// TIA Portal V17 export
// export: Created 2025-04-25T10:07:02.8968061Z, ExportSetting WithDefaults, DisplayName Totally Integrated Automation Portal, DisplayVersion V17 Update 8, DisplayName TIA Portal Openness, DisplayVersion V17 Update 8, DisplayName TIA Portal Version Control Interface, DisplayVersion V17, DisplayName SINAMICS Startdrive Advanced, DisplayVersion V17 SP2, DisplayName SINAMICS Startdrive G110M, G120, G120C, G120D, G120P, G115D, DisplayVersion V17 SP2, DisplayName SINAMICS Startdrive G130, G150, S120, S150, SINAMICS MV, S210, DisplayVersion V17 SP2, DisplayName STEP 7 Professional, DisplayVersion V17 Update 8, DisplayName SINUMERIK ONE STEP 7 Toolbox, DisplayVersion V17 Update 12, DisplayName SINUMERIK 840D sl STEP 7 Toolbox, DisplayVersion V17 Update 12, DisplayName STEP 7 Safety, DisplayVersion V17 Update 6, DisplayName WinCC Advanced / Unified PC, DisplayVersion V17 Update 8
FUNCTION "FC7342_MACHINE_TO_POWDER_PLC_INTERLOCK" : Void   // FC7342, LAD
{ S7_Optimized_Access := 'TRUE' }
VERSION : 0.1
// stored: AutoNumber false, IsIECCheckEnabled false, SetENOAutomatically false, UDAEnableTagReadback false
   VAR_TEMP
      RET_VAL_1 : Int;
   END_VAR
BEGIN

REGION Network 1: LIFE BIT
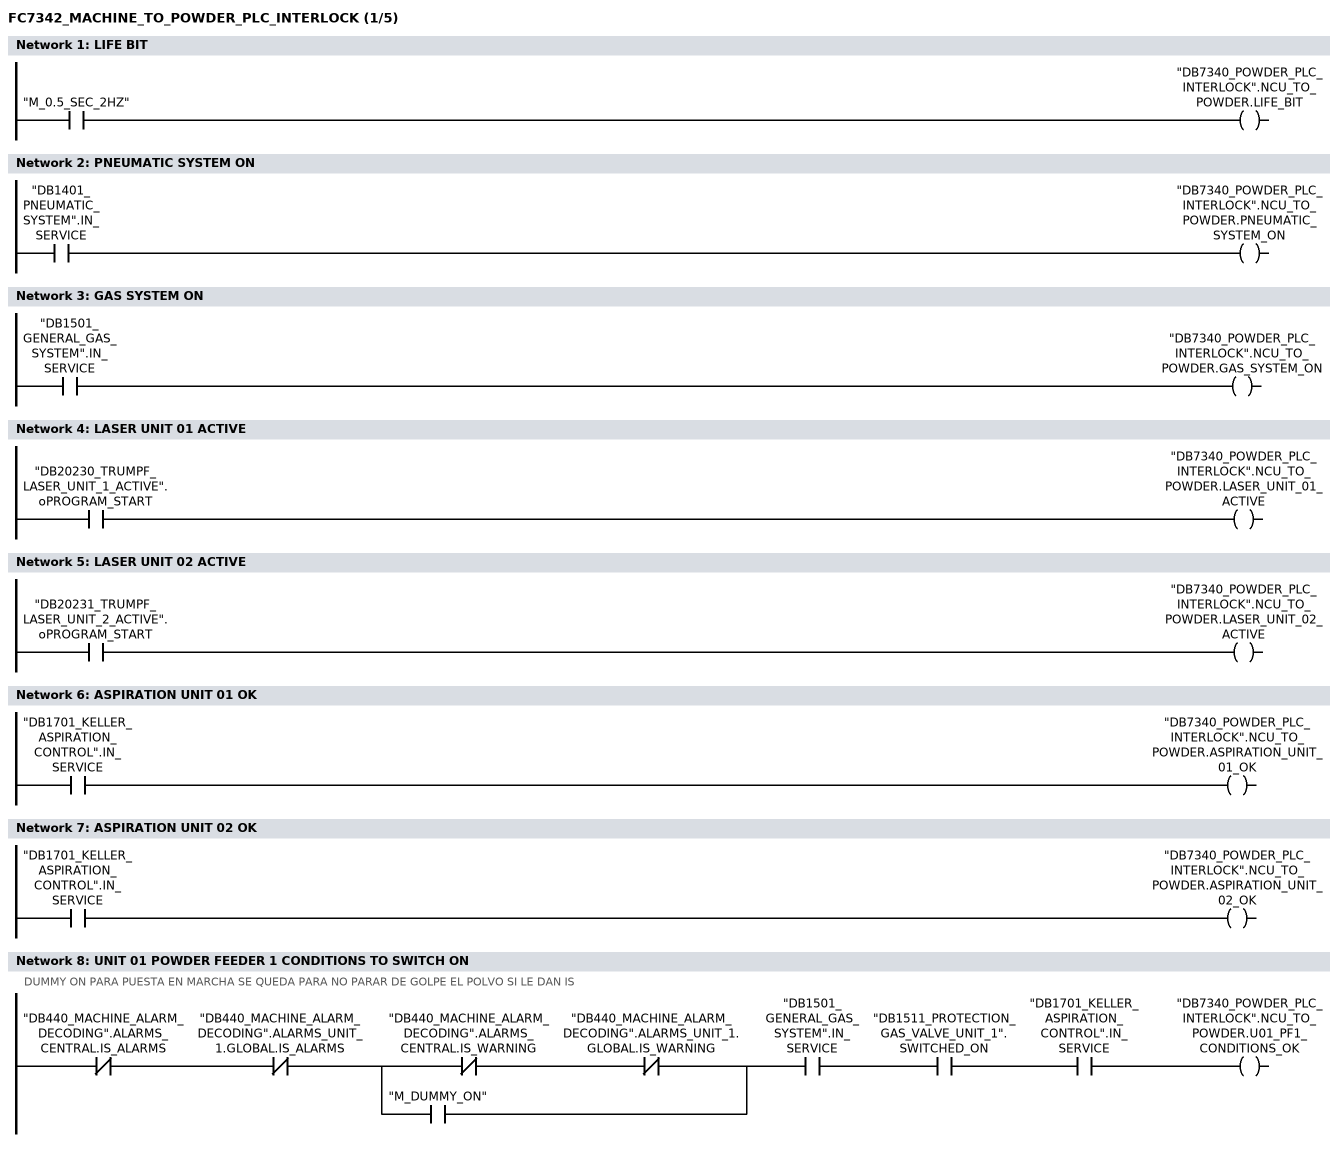
   RUNG wire#powerrail
      Contact( "M_0.5_SEC_2HZ" )
      Coil( "DB7340_POWDER_PLC_INTERLOCK".NCU_TO_POWDER.LIFE_BIT )
   END_RUNG
   // the same network as SCL:
   "DB7340_POWDER_PLC_INTERLOCK".NCU_TO_POWDER.LIFE_BIT := "M_0.5_SEC_2HZ";
END_REGION

REGION Network 2: PNEUMATIC SYSTEM ON
   RUNG wire#powerrail
      Contact( "DB1401_PNEUMATIC_SYSTEM".IN_SERVICE )
      Coil( "DB7340_POWDER_PLC_INTERLOCK".NCU_TO_POWDER.PNEUMATIC_SYSTEM_ON )
   END_RUNG
   // the same network as SCL:
   "DB7340_POWDER_PLC_INTERLOCK".NCU_TO_POWDER.PNEUMATIC_SYSTEM_ON := "DB1401_PNEUMATIC_SYSTEM".IN_SERVICE;
END_REGION

REGION Network 3: GAS SYSTEM ON
   RUNG wire#powerrail
      Contact( "DB1501_GENERAL_GAS_SYSTEM".IN_SERVICE )
      Coil( "DB7340_POWDER_PLC_INTERLOCK".NCU_TO_POWDER.GAS_SYSTEM_ON )
   END_RUNG
   // the same network as SCL:
   "DB7340_POWDER_PLC_INTERLOCK".NCU_TO_POWDER.GAS_SYSTEM_ON := "DB1501_GENERAL_GAS_SYSTEM".IN_SERVICE;
END_REGION

REGION Network 4: LASER UNIT 01 ACTIVE
   RUNG wire#powerrail
      Contact( "DB20230_TRUMPF_LASER_UNIT_1_ACTIVE".oPROGRAM_START )
      Coil( "DB7340_POWDER_PLC_INTERLOCK".NCU_TO_POWDER.LASER_UNIT_01_ACTIVE )
   END_RUNG
   // the same network as SCL:
   "DB7340_POWDER_PLC_INTERLOCK".NCU_TO_POWDER.LASER_UNIT_01_ACTIVE := "DB20230_TRUMPF_LASER_UNIT_1_ACTIVE".oPROGRAM_START;
END_REGION

REGION Network 5: LASER UNIT 02 ACTIVE
   RUNG wire#powerrail
      Contact( "DB20231_TRUMPF_LASER_UNIT_2_ACTIVE".oPROGRAM_START )
      Coil( "DB7340_POWDER_PLC_INTERLOCK".NCU_TO_POWDER.LASER_UNIT_02_ACTIVE )
   END_RUNG
   // the same network as SCL:
   "DB7340_POWDER_PLC_INTERLOCK".NCU_TO_POWDER.LASER_UNIT_02_ACTIVE := "DB20231_TRUMPF_LASER_UNIT_2_ACTIVE".oPROGRAM_START;
END_REGION

REGION Network 6: ASPIRATION UNIT 01 OK
   RUNG wire#powerrail
      Contact( "DB1701_KELLER_ASPIRATION_CONTROL".IN_SERVICE )
      Coil( "DB7340_POWDER_PLC_INTERLOCK".NCU_TO_POWDER.ASPIRATION_UNIT_01_OK )
   END_RUNG
   // the same network as SCL:
   "DB7340_POWDER_PLC_INTERLOCK".NCU_TO_POWDER.ASPIRATION_UNIT_01_OK := "DB1701_KELLER_ASPIRATION_CONTROL".IN_SERVICE;
END_REGION

REGION Network 7: ASPIRATION UNIT 02 OK
   RUNG wire#powerrail
      Contact( "DB1701_KELLER_ASPIRATION_CONTROL".IN_SERVICE )
      Coil( "DB7340_POWDER_PLC_INTERLOCK".NCU_TO_POWDER.ASPIRATION_UNIT_02_OK )
   END_RUNG
   // the same network as SCL:
   "DB7340_POWDER_PLC_INTERLOCK".NCU_TO_POWDER.ASPIRATION_UNIT_02_OK := "DB1701_KELLER_ASPIRATION_CONTROL".IN_SERVICE;
END_REGION

REGION Network 8: UNIT 01 POWDER FEEDER 1 CONDITIONS TO SWITCH ON
   // DUMMY ON PARA PUESTA EN MARCHA SE QUEDA PARA NO PARAR DE GOLPE EL POLVO SI LE DAN IS
   RUNG wire#powerrail
      I_Contact( "DB440_MACHINE_ALARM_DECODING".ALARMS_CENTRAL.IS_ALARMS )
      I_Contact( "DB440_MACHINE_ALARM_DECODING".ALARMS_UNIT_1.GLOBAL.IS_ALARMS )
      wire#w1
      I_Contact( "DB440_MACHINE_ALARM_DECODING".ALARMS_CENTRAL.IS_WARNING )
      I_Contact( "DB440_MACHINE_ALARM_DECODING".ALARMS_UNIT_1.GLOBAL.IS_WARNING )
      wire#w2
      Contact( "DB1501_GENERAL_GAS_SYSTEM".IN_SERVICE )
      Contact( "DB1511_PROTECTION_GAS_VALVE_UNIT_1".SWITCHED_ON )
      Contact( "DB1701_KELLER_ASPIRATION_CONTROL".IN_SERVICE )
      Coil( "DB7340_POWDER_PLC_INTERLOCK".NCU_TO_POWDER.U01_PF1_CONDITIONS_OK )
   END_RUNG
   RUNG wire#w1
      Contact( "M_DUMMY_ON" )
   END_RUNG wire#w2
   // the same network as SCL:
   "DB7340_POWDER_PLC_INTERLOCK".NCU_TO_POWDER.U01_PF1_CONDITIONS_OK := NOT "DB440_MACHINE_ALARM_DECODING".ALARMS_CENTRAL.IS_ALARMS AND NOT "DB440_MACHINE_ALARM_DECODING".ALARMS_UNIT_1.GLOBAL.IS_ALARMS AND ((NOT "DB440_MACHINE_ALARM_DECODING".ALARMS_CENTRAL.IS_WARNING AND NOT "DB440_MACHINE_ALARM_DECODING".ALARMS_UNIT_1.GLOBAL.IS_WARNING) OR "M_DUMMY_ON") AND "DB1501_GENERAL_GAS_SYSTEM".IN_SERVICE AND "DB1511_PROTECTION_GAS_VALVE_UNIT_1".SWITCHED_ON AND "DB1701_KELLER_ASPIRATION_CONTROL".IN_SERVICE;
END_REGION

REGION Network 9: UNIT 02 POWDER FEEDER 1 CONDITIONS TO SWITCH ON
   // DUMMY ON PARA PUESTA EN MARCHA SE QUEDA PARA NO PARAR DE GOLPE EL POLVO SI LE DAN IS
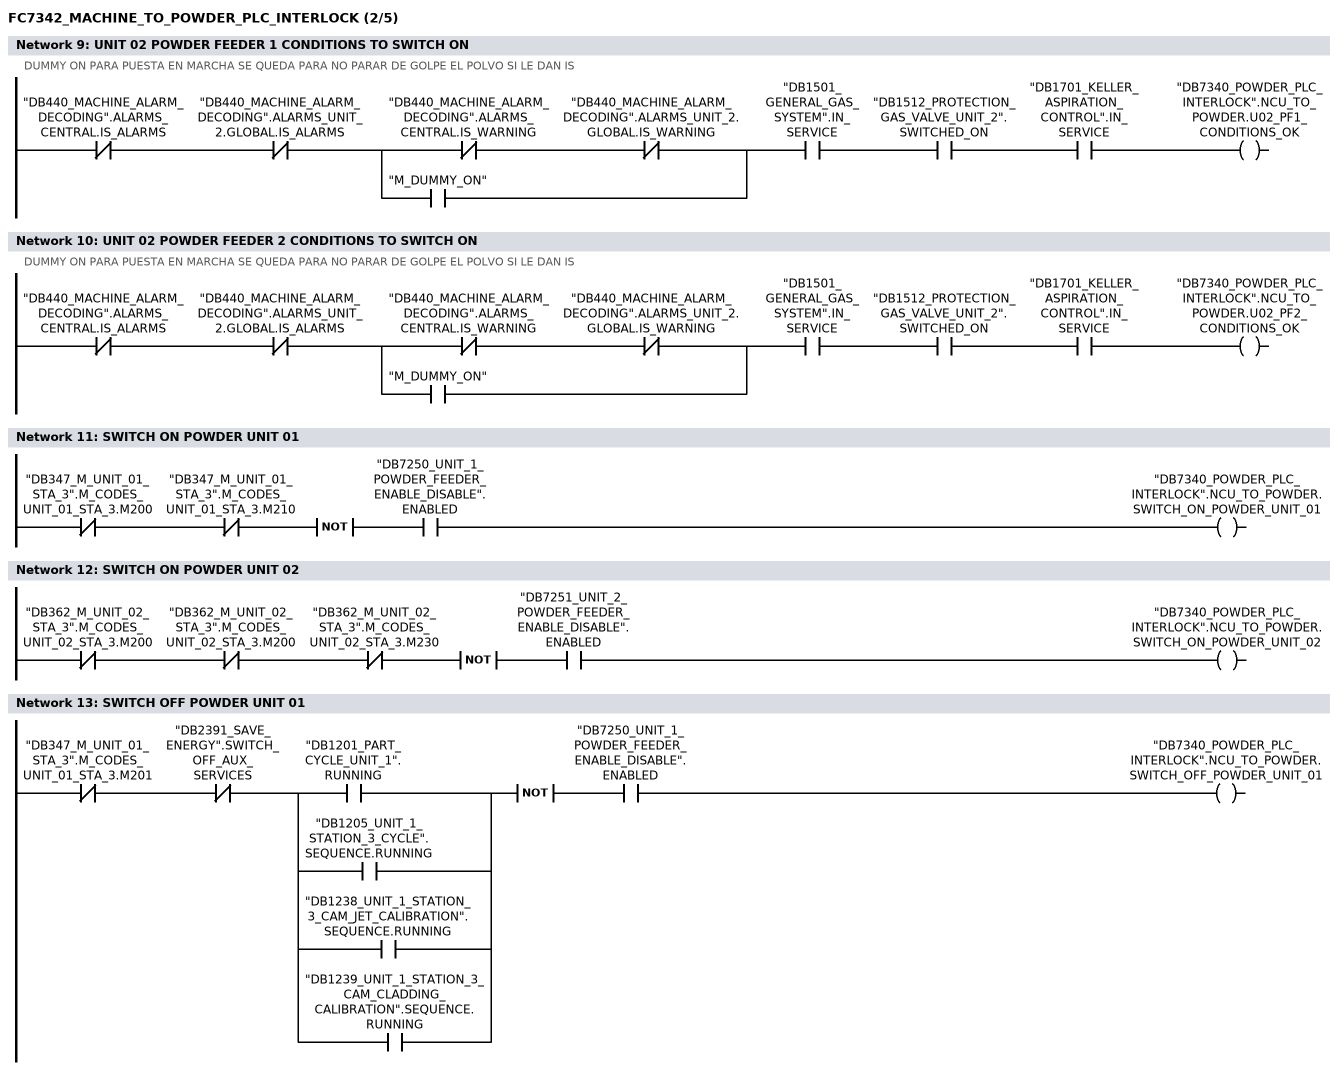
   RUNG wire#powerrail
      I_Contact( "DB440_MACHINE_ALARM_DECODING".ALARMS_CENTRAL.IS_ALARMS )
      I_Contact( "DB440_MACHINE_ALARM_DECODING".ALARMS_UNIT_2.GLOBAL.IS_ALARMS )
      wire#w1
      I_Contact( "DB440_MACHINE_ALARM_DECODING".ALARMS_CENTRAL.IS_WARNING )
      I_Contact( "DB440_MACHINE_ALARM_DECODING".ALARMS_UNIT_2.GLOBAL.IS_WARNING )
      wire#w2
      Contact( "DB1501_GENERAL_GAS_SYSTEM".IN_SERVICE )
      Contact( "DB1512_PROTECTION_GAS_VALVE_UNIT_2".SWITCHED_ON )
      Contact( "DB1701_KELLER_ASPIRATION_CONTROL".IN_SERVICE )
      Coil( "DB7340_POWDER_PLC_INTERLOCK".NCU_TO_POWDER.U02_PF1_CONDITIONS_OK )
   END_RUNG
   RUNG wire#w1
      Contact( "M_DUMMY_ON" )
   END_RUNG wire#w2
   // the same network as SCL:
   "DB7340_POWDER_PLC_INTERLOCK".NCU_TO_POWDER.U02_PF1_CONDITIONS_OK := NOT "DB440_MACHINE_ALARM_DECODING".ALARMS_CENTRAL.IS_ALARMS AND NOT "DB440_MACHINE_ALARM_DECODING".ALARMS_UNIT_2.GLOBAL.IS_ALARMS AND ((NOT "DB440_MACHINE_ALARM_DECODING".ALARMS_CENTRAL.IS_WARNING AND NOT "DB440_MACHINE_ALARM_DECODING".ALARMS_UNIT_2.GLOBAL.IS_WARNING) OR "M_DUMMY_ON") AND "DB1501_GENERAL_GAS_SYSTEM".IN_SERVICE AND "DB1512_PROTECTION_GAS_VALVE_UNIT_2".SWITCHED_ON AND "DB1701_KELLER_ASPIRATION_CONTROL".IN_SERVICE;
END_REGION

REGION Network 10: UNIT 02 POWDER FEEDER 2 CONDITIONS TO SWITCH ON
   // DUMMY ON PARA PUESTA EN MARCHA SE QUEDA PARA NO PARAR DE GOLPE EL POLVO SI LE DAN IS
   RUNG wire#powerrail
      I_Contact( "DB440_MACHINE_ALARM_DECODING".ALARMS_CENTRAL.IS_ALARMS )
      I_Contact( "DB440_MACHINE_ALARM_DECODING".ALARMS_UNIT_2.GLOBAL.IS_ALARMS )
      wire#w1
      I_Contact( "DB440_MACHINE_ALARM_DECODING".ALARMS_CENTRAL.IS_WARNING )
      I_Contact( "DB440_MACHINE_ALARM_DECODING".ALARMS_UNIT_2.GLOBAL.IS_WARNING )
      wire#w2
      Contact( "DB1501_GENERAL_GAS_SYSTEM".IN_SERVICE )
      Contact( "DB1512_PROTECTION_GAS_VALVE_UNIT_2".SWITCHED_ON )
      Contact( "DB1701_KELLER_ASPIRATION_CONTROL".IN_SERVICE )
      Coil( "DB7340_POWDER_PLC_INTERLOCK".NCU_TO_POWDER.U02_PF2_CONDITIONS_OK )
   END_RUNG
   RUNG wire#w1
      Contact( "M_DUMMY_ON" )
   END_RUNG wire#w2
   // the same network as SCL:
   "DB7340_POWDER_PLC_INTERLOCK".NCU_TO_POWDER.U02_PF2_CONDITIONS_OK := NOT "DB440_MACHINE_ALARM_DECODING".ALARMS_CENTRAL.IS_ALARMS AND NOT "DB440_MACHINE_ALARM_DECODING".ALARMS_UNIT_2.GLOBAL.IS_ALARMS AND ((NOT "DB440_MACHINE_ALARM_DECODING".ALARMS_CENTRAL.IS_WARNING AND NOT "DB440_MACHINE_ALARM_DECODING".ALARMS_UNIT_2.GLOBAL.IS_WARNING) OR "M_DUMMY_ON") AND "DB1501_GENERAL_GAS_SYSTEM".IN_SERVICE AND "DB1512_PROTECTION_GAS_VALVE_UNIT_2".SWITCHED_ON AND "DB1701_KELLER_ASPIRATION_CONTROL".IN_SERVICE;
END_REGION

REGION Network 11: SWITCH ON POWDER UNIT 01
   RUNG wire#powerrail
      I_Contact( "DB347_M_UNIT_01_STA_3".M_CODES_UNIT_01_STA_3.M200 )
      I_Contact( "DB347_M_UNIT_01_STA_3".M_CODES_UNIT_01_STA_3.M210 )
      Not()
      Contact( "DB7250_UNIT_1_POWDER_FEEDER_ENABLE_DISABLE".ENABLED )
      Coil( "DB7340_POWDER_PLC_INTERLOCK".NCU_TO_POWDER.SWITCH_ON_POWDER_UNIT_01 )
   END_RUNG
   // the same network as SCL:
   "DB7340_POWDER_PLC_INTERLOCK".NCU_TO_POWDER.SWITCH_ON_POWDER_UNIT_01 := NOT (NOT "DB347_M_UNIT_01_STA_3".M_CODES_UNIT_01_STA_3.M200 AND NOT "DB347_M_UNIT_01_STA_3".M_CODES_UNIT_01_STA_3.M210) AND "DB7250_UNIT_1_POWDER_FEEDER_ENABLE_DISABLE".ENABLED;
END_REGION

REGION Network 12: SWITCH ON POWDER UNIT 02
   RUNG wire#powerrail
      I_Contact( "DB362_M_UNIT_02_STA_3".M_CODES_UNIT_02_STA_3.M200 )
      I_Contact( "DB362_M_UNIT_02_STA_3".M_CODES_UNIT_02_STA_3.M200 )
      I_Contact( "DB362_M_UNIT_02_STA_3".M_CODES_UNIT_02_STA_3.M230 )
      Not()
      Contact( "DB7251_UNIT_2_POWDER_FEEDER_ENABLE_DISABLE".ENABLED )
      Coil( "DB7340_POWDER_PLC_INTERLOCK".NCU_TO_POWDER.SWITCH_ON_POWDER_UNIT_02 )
   END_RUNG
   // the same network as SCL:
   "DB7340_POWDER_PLC_INTERLOCK".NCU_TO_POWDER.SWITCH_ON_POWDER_UNIT_02 := NOT (NOT "DB362_M_UNIT_02_STA_3".M_CODES_UNIT_02_STA_3.M200 AND NOT "DB362_M_UNIT_02_STA_3".M_CODES_UNIT_02_STA_3.M200 AND NOT "DB362_M_UNIT_02_STA_3".M_CODES_UNIT_02_STA_3.M230) AND "DB7251_UNIT_2_POWDER_FEEDER_ENABLE_DISABLE".ENABLED;
END_REGION

REGION Network 13: SWITCH OFF POWDER UNIT 01
   RUNG wire#powerrail
      I_Contact( "DB347_M_UNIT_01_STA_3".M_CODES_UNIT_01_STA_3.M201 )
      I_Contact( "DB2391_SAVE_ENERGY".SWITCH_OFF_AUX_SERVICES )
      wire#w1
      Contact( "DB1201_PART_CYCLE_UNIT_1".RUNNING )
      wire#w2
      Not()
      Contact( "DB7250_UNIT_1_POWDER_FEEDER_ENABLE_DISABLE".ENABLED )
      Coil( "DB7340_POWDER_PLC_INTERLOCK".NCU_TO_POWDER.SWITCH_OFF_POWDER_UNIT_01 )
   END_RUNG
   RUNG wire#w1
      Contact( "DB1205_UNIT_1_STATION_3_CYCLE".SEQUENCE.RUNNING )
   END_RUNG wire#w2
   RUNG wire#w1
      Contact( "DB1238_UNIT_1_STATION_3_CAM_JET_CALIBRATION".SEQUENCE.RUNNING )
   END_RUNG wire#w2
   RUNG wire#w1
      Contact( "DB1239_UNIT_1_STATION_3_CAM_CLADDING_CALIBRATION".SEQUENCE.RUNNING )
   END_RUNG wire#w2
   // the same network as SCL:
   "DB7340_POWDER_PLC_INTERLOCK".NCU_TO_POWDER.SWITCH_OFF_POWDER_UNIT_01 := NOT (NOT "DB347_M_UNIT_01_STA_3".M_CODES_UNIT_01_STA_3.M201 AND NOT "DB2391_SAVE_ENERGY".SWITCH_OFF_AUX_SERVICES AND ("DB1201_PART_CYCLE_UNIT_1".RUNNING OR "DB1205_UNIT_1_STATION_3_CYCLE".SEQUENCE.RUNNING OR "DB1238_UNIT_1_STATION_3_CAM_JET_CALIBRATION".SEQUENCE.RUNNING OR "DB1239_UNIT_1_STATION_3_CAM_CLADDING_CALIBRATION".SEQUENCE.RUNNING)) AND "DB7250_UNIT_1_POWDER_FEEDER_ENABLE_DISABLE".ENABLED;
END_REGION

REGION Network 14: SWITCH OFF POWDER UNIT 02
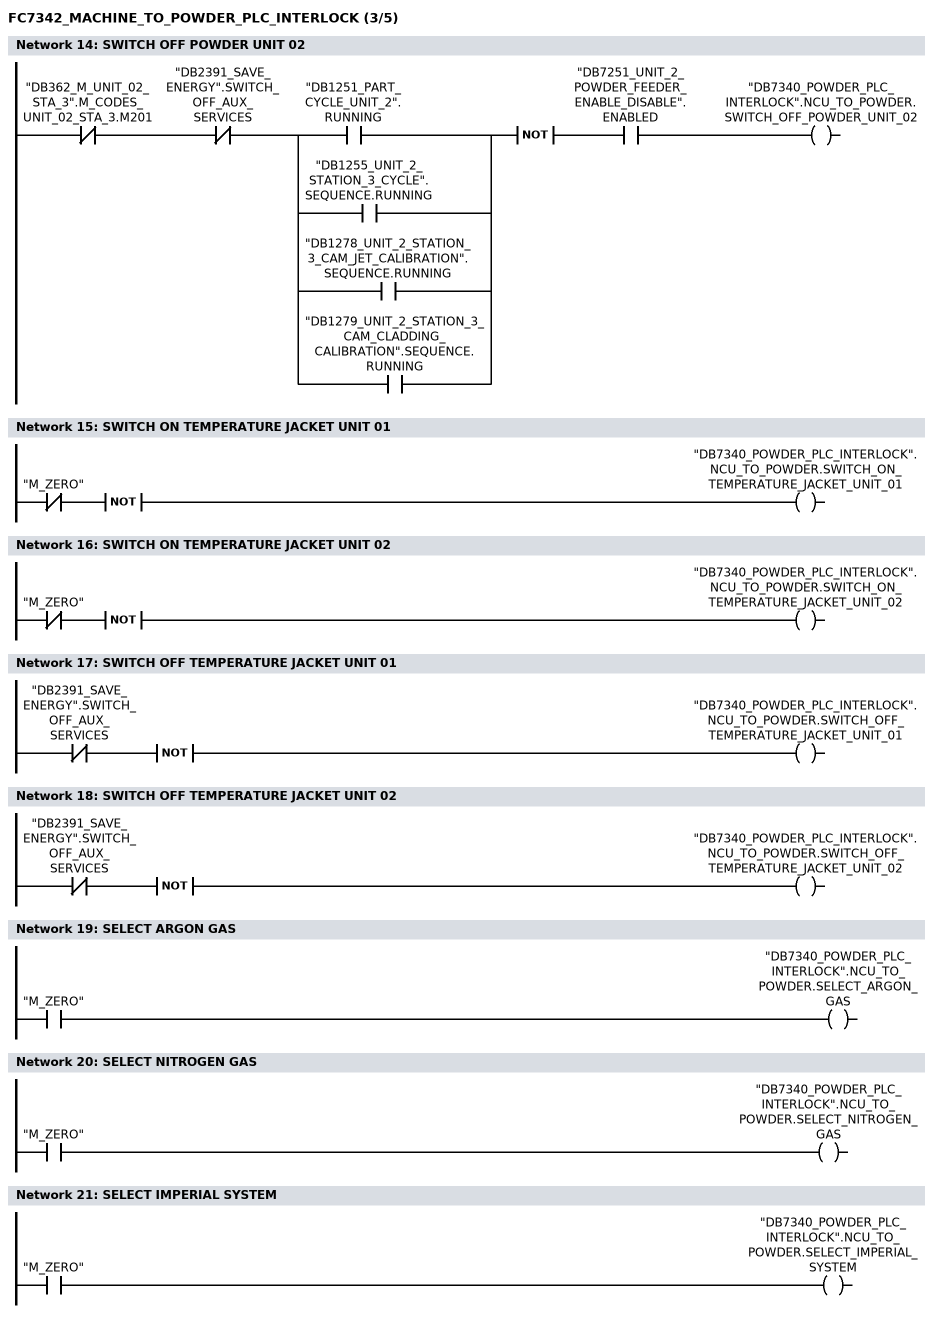
   RUNG wire#powerrail
      I_Contact( "DB362_M_UNIT_02_STA_3".M_CODES_UNIT_02_STA_3.M201 )
      I_Contact( "DB2391_SAVE_ENERGY".SWITCH_OFF_AUX_SERVICES )
      wire#w1
      Contact( "DB1251_PART_CYCLE_UNIT_2".RUNNING )
      wire#w2
      Not()
      Contact( "DB7251_UNIT_2_POWDER_FEEDER_ENABLE_DISABLE".ENABLED )
      Coil( "DB7340_POWDER_PLC_INTERLOCK".NCU_TO_POWDER.SWITCH_OFF_POWDER_UNIT_02 )
   END_RUNG
   RUNG wire#w1
      Contact( "DB1255_UNIT_2_STATION_3_CYCLE".SEQUENCE.RUNNING )
   END_RUNG wire#w2
   RUNG wire#w1
      Contact( "DB1278_UNIT_2_STATION_3_CAM_JET_CALIBRATION".SEQUENCE.RUNNING )
   END_RUNG wire#w2
   RUNG wire#w1
      Contact( "DB1279_UNIT_2_STATION_3_CAM_CLADDING_CALIBRATION".SEQUENCE.RUNNING )
   END_RUNG wire#w2
   // the same network as SCL:
   "DB7340_POWDER_PLC_INTERLOCK".NCU_TO_POWDER.SWITCH_OFF_POWDER_UNIT_02 := NOT (NOT "DB362_M_UNIT_02_STA_3".M_CODES_UNIT_02_STA_3.M201 AND NOT "DB2391_SAVE_ENERGY".SWITCH_OFF_AUX_SERVICES AND ("DB1251_PART_CYCLE_UNIT_2".RUNNING OR "DB1255_UNIT_2_STATION_3_CYCLE".SEQUENCE.RUNNING OR "DB1278_UNIT_2_STATION_3_CAM_JET_CALIBRATION".SEQUENCE.RUNNING OR "DB1279_UNIT_2_STATION_3_CAM_CLADDING_CALIBRATION".SEQUENCE.RUNNING)) AND "DB7251_UNIT_2_POWDER_FEEDER_ENABLE_DISABLE".ENABLED;
END_REGION

REGION Network 15: SWITCH ON TEMPERATURE JACKET UNIT 01
   RUNG wire#powerrail
      I_Contact( "M_ZERO" )
      Not()
      Coil( "DB7340_POWDER_PLC_INTERLOCK".NCU_TO_POWDER.SWITCH_ON_TEMPERATURE_JACKET_UNIT_01 )
   END_RUNG
   // the same network as SCL:
   "DB7340_POWDER_PLC_INTERLOCK".NCU_TO_POWDER.SWITCH_ON_TEMPERATURE_JACKET_UNIT_01 := NOT (NOT "M_ZERO");
END_REGION

REGION Network 16: SWITCH ON TEMPERATURE JACKET UNIT 02
   RUNG wire#powerrail
      I_Contact( "M_ZERO" )
      Not()
      Coil( "DB7340_POWDER_PLC_INTERLOCK".NCU_TO_POWDER.SWITCH_ON_TEMPERATURE_JACKET_UNIT_02 )
   END_RUNG
   // the same network as SCL:
   "DB7340_POWDER_PLC_INTERLOCK".NCU_TO_POWDER.SWITCH_ON_TEMPERATURE_JACKET_UNIT_02 := NOT (NOT "M_ZERO");
END_REGION

REGION Network 17: SWITCH OFF TEMPERATURE JACKET UNIT 01
   RUNG wire#powerrail
      I_Contact( "DB2391_SAVE_ENERGY".SWITCH_OFF_AUX_SERVICES )
      Not()
      Coil( "DB7340_POWDER_PLC_INTERLOCK".NCU_TO_POWDER.SWITCH_OFF_TEMPERATURE_JACKET_UNIT_01 )
   END_RUNG
   // the same network as SCL:
   "DB7340_POWDER_PLC_INTERLOCK".NCU_TO_POWDER.SWITCH_OFF_TEMPERATURE_JACKET_UNIT_01 := NOT (NOT "DB2391_SAVE_ENERGY".SWITCH_OFF_AUX_SERVICES);
END_REGION

REGION Network 18: SWITCH OFF TEMPERATURE JACKET UNIT 02
   RUNG wire#powerrail
      I_Contact( "DB2391_SAVE_ENERGY".SWITCH_OFF_AUX_SERVICES )
      Not()
      Coil( "DB7340_POWDER_PLC_INTERLOCK".NCU_TO_POWDER.SWITCH_OFF_TEMPERATURE_JACKET_UNIT_02 )
   END_RUNG
   // the same network as SCL:
   "DB7340_POWDER_PLC_INTERLOCK".NCU_TO_POWDER.SWITCH_OFF_TEMPERATURE_JACKET_UNIT_02 := NOT (NOT "DB2391_SAVE_ENERGY".SWITCH_OFF_AUX_SERVICES);
END_REGION

REGION Network 19: SELECT ARGON GAS
   RUNG wire#powerrail
      Contact( "M_ZERO" )
      Coil( "DB7340_POWDER_PLC_INTERLOCK".NCU_TO_POWDER.SELECT_ARGON_GAS )
   END_RUNG
   // the same network as SCL:
   "DB7340_POWDER_PLC_INTERLOCK".NCU_TO_POWDER.SELECT_ARGON_GAS := "M_ZERO";
END_REGION

REGION Network 20: SELECT NITROGEN GAS
   RUNG wire#powerrail
      Contact( "M_ZERO" )
      Coil( "DB7340_POWDER_PLC_INTERLOCK".NCU_TO_POWDER.SELECT_NITROGEN_GAS )
   END_RUNG
   // the same network as SCL:
   "DB7340_POWDER_PLC_INTERLOCK".NCU_TO_POWDER.SELECT_NITROGEN_GAS := "M_ZERO";
END_REGION

REGION Network 21: SELECT IMPERIAL SYSTEM
   RUNG wire#powerrail
      Contact( "M_ZERO" )
      Coil( "DB7340_POWDER_PLC_INTERLOCK".NCU_TO_POWDER.SELECT_IMPERIAL_SYSTEM )
   END_RUNG
   // the same network as SCL:
   "DB7340_POWDER_PLC_INTERLOCK".NCU_TO_POWDER.SELECT_IMPERIAL_SYSTEM := "M_ZERO";
END_REGION

REGION Network 22: SELECT METRIC SYSTEM
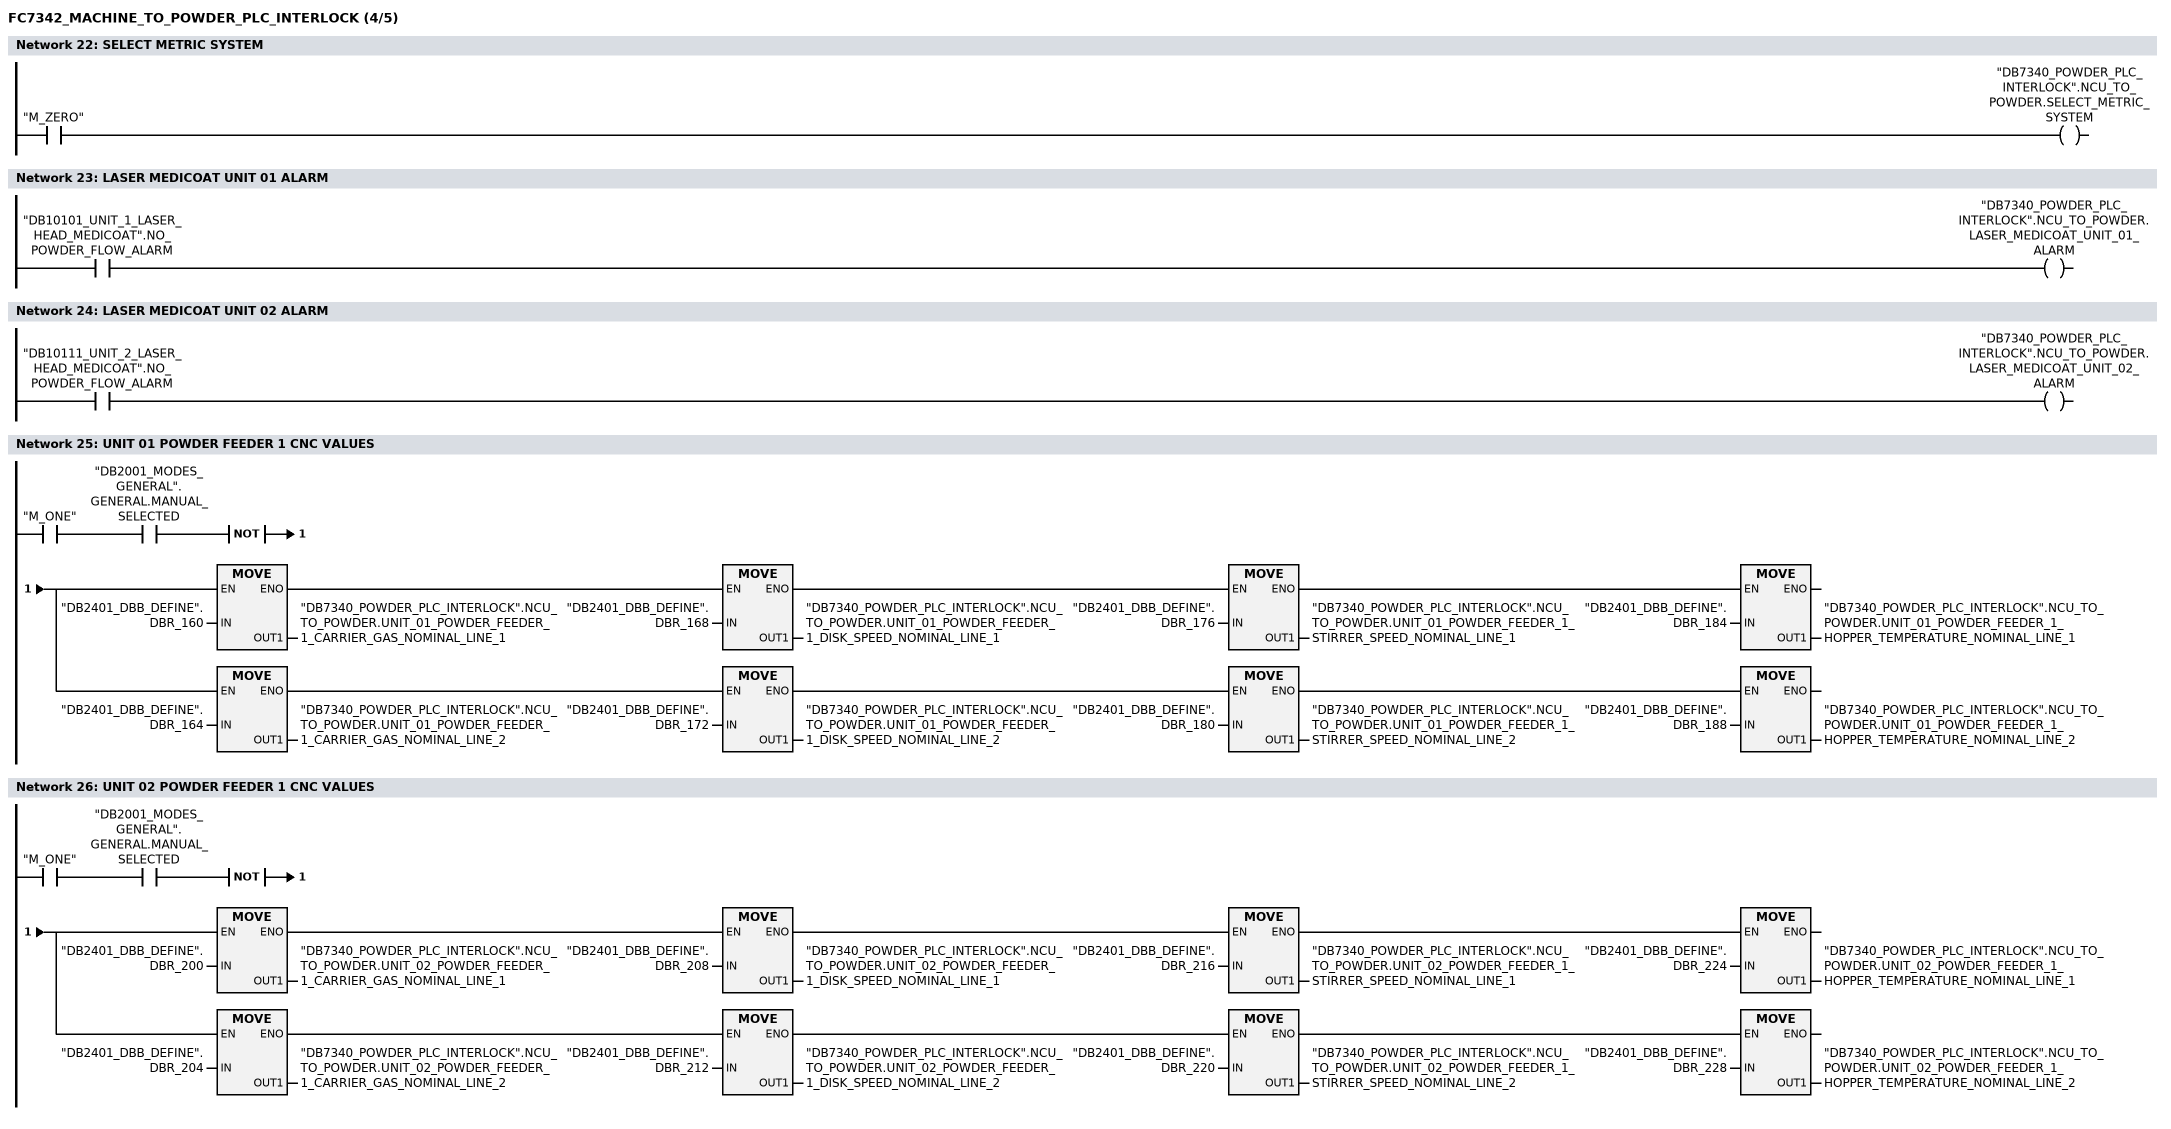
   RUNG wire#powerrail
      Contact( "M_ZERO" )
      Coil( "DB7340_POWDER_PLC_INTERLOCK".NCU_TO_POWDER.SELECT_METRIC_SYSTEM )
   END_RUNG
   // the same network as SCL:
   "DB7340_POWDER_PLC_INTERLOCK".NCU_TO_POWDER.SELECT_METRIC_SYSTEM := "M_ZERO";
END_REGION

REGION Network 23: LASER MEDICOAT UNIT 01 ALARM
   RUNG wire#powerrail
      Contact( "DB10101_UNIT_1_LASER_HEAD_MEDICOAT".NO_POWDER_FLOW_ALARM )
      Coil( "DB7340_POWDER_PLC_INTERLOCK".NCU_TO_POWDER.LASER_MEDICOAT_UNIT_01_ALARM )
   END_RUNG
   // the same network as SCL:
   "DB7340_POWDER_PLC_INTERLOCK".NCU_TO_POWDER.LASER_MEDICOAT_UNIT_01_ALARM := "DB10101_UNIT_1_LASER_HEAD_MEDICOAT".NO_POWDER_FLOW_ALARM;
END_REGION

REGION Network 24: LASER MEDICOAT UNIT 02 ALARM
   RUNG wire#powerrail
      Contact( "DB10111_UNIT_2_LASER_HEAD_MEDICOAT".NO_POWDER_FLOW_ALARM )
      Coil( "DB7340_POWDER_PLC_INTERLOCK".NCU_TO_POWDER.LASER_MEDICOAT_UNIT_02_ALARM )
   END_RUNG
   // the same network as SCL:
   "DB7340_POWDER_PLC_INTERLOCK".NCU_TO_POWDER.LASER_MEDICOAT_UNIT_02_ALARM := "DB10111_UNIT_2_LASER_HEAD_MEDICOAT".NO_POWDER_FLOW_ALARM;
END_REGION

REGION Network 25: UNIT 01 POWDER FEEDER 1 CNC VALUES
   RUNG wire#powerrail
      Contact( "M_ONE" )
      Contact( "DB2001_MODES_GENERAL".GENERAL.MANUAL_SELECTED )
      Not()
      wire#w1
      Move(in := "DB2401_DBB_DEFINE".DBR_160, out1 => "DB7340_POWDER_PLC_INTERLOCK".NCU_TO_POWDER.UNIT_01_POWDER_FEEDER_1_CARRIER_GAS_NOMINAL_LINE_1)
      Move(in := "DB2401_DBB_DEFINE".DBR_168, out1 => "DB7340_POWDER_PLC_INTERLOCK".NCU_TO_POWDER.UNIT_01_POWDER_FEEDER_1_DISK_SPEED_NOMINAL_LINE_1)
      Move(in := "DB2401_DBB_DEFINE".DBR_176, out1 => "DB7340_POWDER_PLC_INTERLOCK".NCU_TO_POWDER.UNIT_01_POWDER_FEEDER_1_STIRRER_SPEED_NOMINAL_LINE_1)
      Move(in := "DB2401_DBB_DEFINE".DBR_184, out1 => "DB7340_POWDER_PLC_INTERLOCK".NCU_TO_POWDER.UNIT_01_POWDER_FEEDER_1_HOPPER_TEMPERATURE_NOMINAL_LINE_1)
   END_RUNG
   RUNG wire#w1
      Move(in := "DB2401_DBB_DEFINE".DBR_164, out1 => "DB7340_POWDER_PLC_INTERLOCK".NCU_TO_POWDER.UNIT_01_POWDER_FEEDER_1_CARRIER_GAS_NOMINAL_LINE_2)
      Move(in := "DB2401_DBB_DEFINE".DBR_172, out1 => "DB7340_POWDER_PLC_INTERLOCK".NCU_TO_POWDER.UNIT_01_POWDER_FEEDER_1_DISK_SPEED_NOMINAL_LINE_2)
      Move(in := "DB2401_DBB_DEFINE".DBR_180, out1 => "DB7340_POWDER_PLC_INTERLOCK".NCU_TO_POWDER.UNIT_01_POWDER_FEEDER_1_STIRRER_SPEED_NOMINAL_LINE_2)
      Move(in := "DB2401_DBB_DEFINE".DBR_188, out1 => "DB7340_POWDER_PLC_INTERLOCK".NCU_TO_POWDER.UNIT_01_POWDER_FEEDER_1_HOPPER_TEMPERATURE_NOMINAL_LINE_2)
   END_RUNG
   // the same network as SCL:
   IF NOT ("M_ONE" AND "DB2001_MODES_GENERAL".GENERAL.MANUAL_SELECTED) THEN
       "DB7340_POWDER_PLC_INTERLOCK".NCU_TO_POWDER.UNIT_01_POWDER_FEEDER_1_CARRIER_GAS_NOMINAL_LINE_1 := "DB2401_DBB_DEFINE".DBR_160;
       "DB7340_POWDER_PLC_INTERLOCK".NCU_TO_POWDER.UNIT_01_POWDER_FEEDER_1_DISK_SPEED_NOMINAL_LINE_1 := "DB2401_DBB_DEFINE".DBR_168;
       "DB7340_POWDER_PLC_INTERLOCK".NCU_TO_POWDER.UNIT_01_POWDER_FEEDER_1_STIRRER_SPEED_NOMINAL_LINE_1 := "DB2401_DBB_DEFINE".DBR_176;
       "DB7340_POWDER_PLC_INTERLOCK".NCU_TO_POWDER.UNIT_01_POWDER_FEEDER_1_HOPPER_TEMPERATURE_NOMINAL_LINE_1 := "DB2401_DBB_DEFINE".DBR_184;
       "DB7340_POWDER_PLC_INTERLOCK".NCU_TO_POWDER.UNIT_01_POWDER_FEEDER_1_CARRIER_GAS_NOMINAL_LINE_2 := "DB2401_DBB_DEFINE".DBR_164;
       "DB7340_POWDER_PLC_INTERLOCK".NCU_TO_POWDER.UNIT_01_POWDER_FEEDER_1_DISK_SPEED_NOMINAL_LINE_2 := "DB2401_DBB_DEFINE".DBR_172;
       "DB7340_POWDER_PLC_INTERLOCK".NCU_TO_POWDER.UNIT_01_POWDER_FEEDER_1_STIRRER_SPEED_NOMINAL_LINE_2 := "DB2401_DBB_DEFINE".DBR_180;
       "DB7340_POWDER_PLC_INTERLOCK".NCU_TO_POWDER.UNIT_01_POWDER_FEEDER_1_HOPPER_TEMPERATURE_NOMINAL_LINE_2 := "DB2401_DBB_DEFINE".DBR_188;
   END_IF;
END_REGION

REGION Network 26: UNIT 02 POWDER FEEDER 1 CNC VALUES
   RUNG wire#powerrail
      Contact( "M_ONE" )
      Contact( "DB2001_MODES_GENERAL".GENERAL.MANUAL_SELECTED )
      Not()
      wire#w1
      Move(in := "DB2401_DBB_DEFINE".DBR_200, out1 => "DB7340_POWDER_PLC_INTERLOCK".NCU_TO_POWDER.UNIT_02_POWDER_FEEDER_1_CARRIER_GAS_NOMINAL_LINE_1)
      Move(in := "DB2401_DBB_DEFINE".DBR_208, out1 => "DB7340_POWDER_PLC_INTERLOCK".NCU_TO_POWDER.UNIT_02_POWDER_FEEDER_1_DISK_SPEED_NOMINAL_LINE_1)
      Move(in := "DB2401_DBB_DEFINE".DBR_216, out1 => "DB7340_POWDER_PLC_INTERLOCK".NCU_TO_POWDER.UNIT_02_POWDER_FEEDER_1_STIRRER_SPEED_NOMINAL_LINE_1)
      Move(in := "DB2401_DBB_DEFINE".DBR_224, out1 => "DB7340_POWDER_PLC_INTERLOCK".NCU_TO_POWDER.UNIT_02_POWDER_FEEDER_1_HOPPER_TEMPERATURE_NOMINAL_LINE_1)
   END_RUNG
   RUNG wire#w1
      Move(in := "DB2401_DBB_DEFINE".DBR_204, out1 => "DB7340_POWDER_PLC_INTERLOCK".NCU_TO_POWDER.UNIT_02_POWDER_FEEDER_1_CARRIER_GAS_NOMINAL_LINE_2)
      Move(in := "DB2401_DBB_DEFINE".DBR_212, out1 => "DB7340_POWDER_PLC_INTERLOCK".NCU_TO_POWDER.UNIT_02_POWDER_FEEDER_1_DISK_SPEED_NOMINAL_LINE_2)
      Move(in := "DB2401_DBB_DEFINE".DBR_220, out1 => "DB7340_POWDER_PLC_INTERLOCK".NCU_TO_POWDER.UNIT_02_POWDER_FEEDER_1_STIRRER_SPEED_NOMINAL_LINE_2)
      Move(in := "DB2401_DBB_DEFINE".DBR_228, out1 => "DB7340_POWDER_PLC_INTERLOCK".NCU_TO_POWDER.UNIT_02_POWDER_FEEDER_1_HOPPER_TEMPERATURE_NOMINAL_LINE_2)
   END_RUNG
   // the same network as SCL:
   IF NOT ("M_ONE" AND "DB2001_MODES_GENERAL".GENERAL.MANUAL_SELECTED) THEN
       "DB7340_POWDER_PLC_INTERLOCK".NCU_TO_POWDER.UNIT_02_POWDER_FEEDER_1_CARRIER_GAS_NOMINAL_LINE_1 := "DB2401_DBB_DEFINE".DBR_200;
       "DB7340_POWDER_PLC_INTERLOCK".NCU_TO_POWDER.UNIT_02_POWDER_FEEDER_1_DISK_SPEED_NOMINAL_LINE_1 := "DB2401_DBB_DEFINE".DBR_208;
       "DB7340_POWDER_PLC_INTERLOCK".NCU_TO_POWDER.UNIT_02_POWDER_FEEDER_1_STIRRER_SPEED_NOMINAL_LINE_1 := "DB2401_DBB_DEFINE".DBR_216;
       "DB7340_POWDER_PLC_INTERLOCK".NCU_TO_POWDER.UNIT_02_POWDER_FEEDER_1_HOPPER_TEMPERATURE_NOMINAL_LINE_1 := "DB2401_DBB_DEFINE".DBR_224;
       "DB7340_POWDER_PLC_INTERLOCK".NCU_TO_POWDER.UNIT_02_POWDER_FEEDER_1_CARRIER_GAS_NOMINAL_LINE_2 := "DB2401_DBB_DEFINE".DBR_204;
       "DB7340_POWDER_PLC_INTERLOCK".NCU_TO_POWDER.UNIT_02_POWDER_FEEDER_1_DISK_SPEED_NOMINAL_LINE_2 := "DB2401_DBB_DEFINE".DBR_212;
       "DB7340_POWDER_PLC_INTERLOCK".NCU_TO_POWDER.UNIT_02_POWDER_FEEDER_1_STIRRER_SPEED_NOMINAL_LINE_2 := "DB2401_DBB_DEFINE".DBR_220;
       "DB7340_POWDER_PLC_INTERLOCK".NCU_TO_POWDER.UNIT_02_POWDER_FEEDER_1_HOPPER_TEMPERATURE_NOMINAL_LINE_2 := "DB2401_DBB_DEFINE".DBR_228;
   END_IF;
END_REGION

REGION Network 27: UNIT 02 POWDER FEEDER 2 CNC VALUES
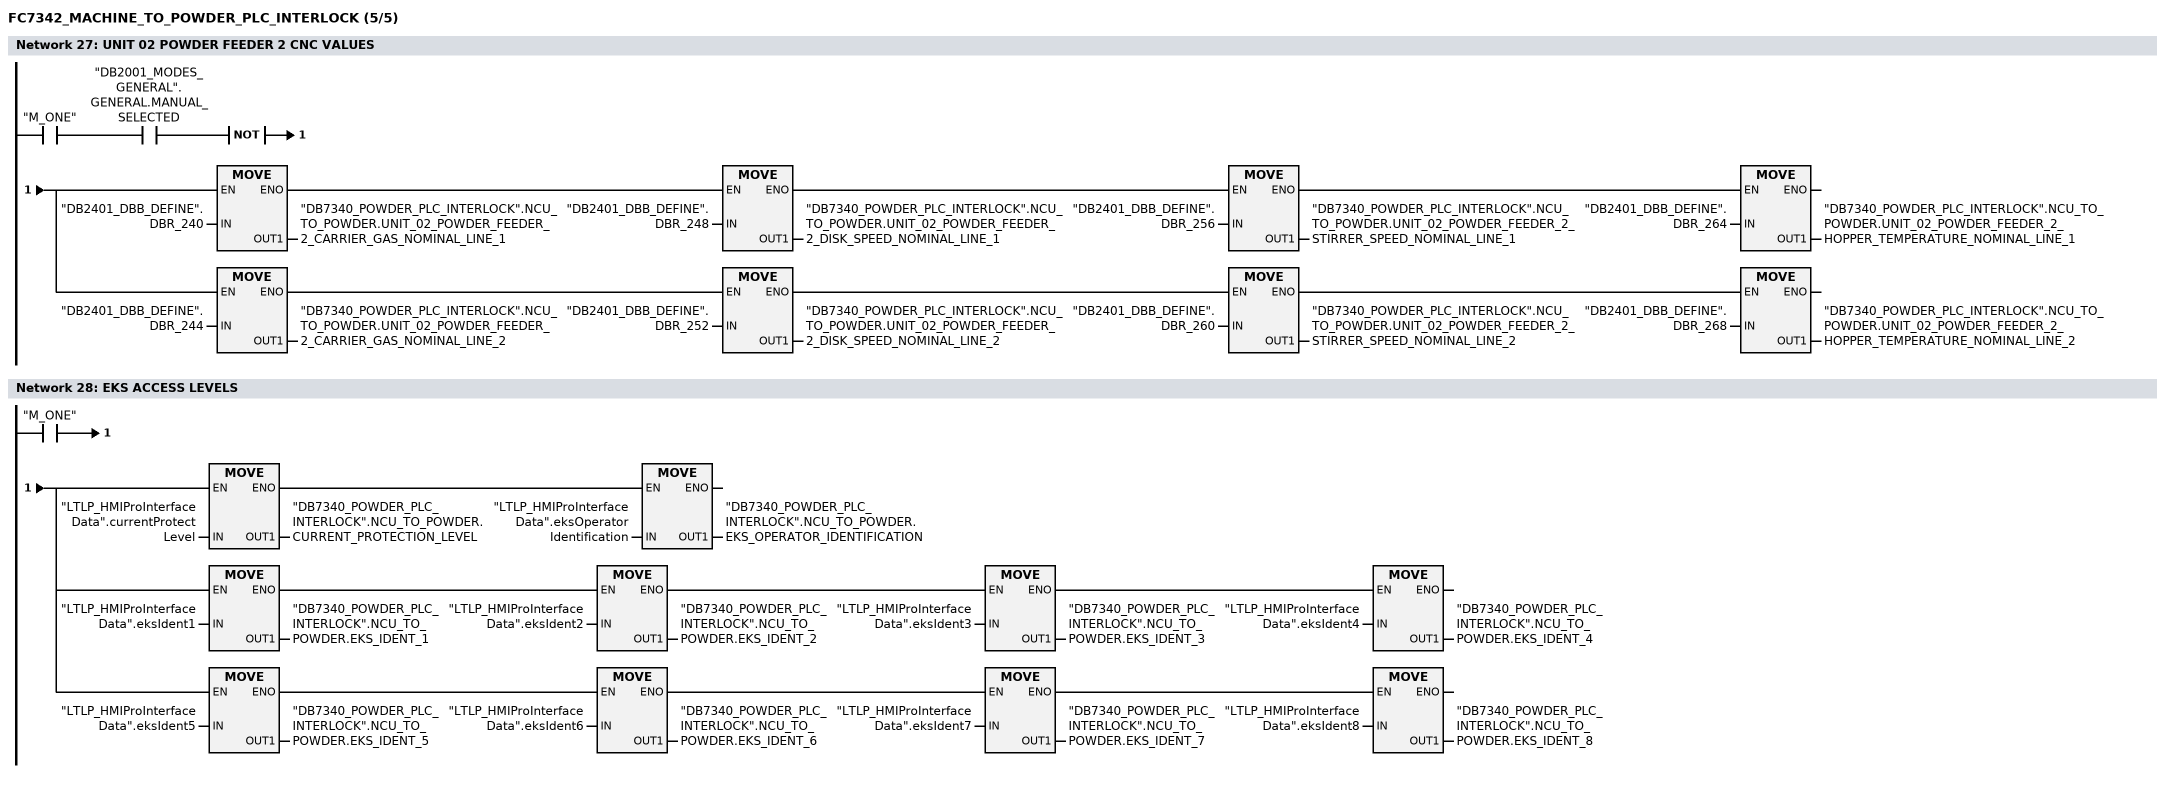
   RUNG wire#powerrail
      Contact( "M_ONE" )
      Contact( "DB2001_MODES_GENERAL".GENERAL.MANUAL_SELECTED )
      Not()
      wire#w1
      Move(in := "DB2401_DBB_DEFINE".DBR_240, out1 => "DB7340_POWDER_PLC_INTERLOCK".NCU_TO_POWDER.UNIT_02_POWDER_FEEDER_2_CARRIER_GAS_NOMINAL_LINE_1)
      Move(in := "DB2401_DBB_DEFINE".DBR_248, out1 => "DB7340_POWDER_PLC_INTERLOCK".NCU_TO_POWDER.UNIT_02_POWDER_FEEDER_2_DISK_SPEED_NOMINAL_LINE_1)
      Move(in := "DB2401_DBB_DEFINE".DBR_256, out1 => "DB7340_POWDER_PLC_INTERLOCK".NCU_TO_POWDER.UNIT_02_POWDER_FEEDER_2_STIRRER_SPEED_NOMINAL_LINE_1)
      Move(in := "DB2401_DBB_DEFINE".DBR_264, out1 => "DB7340_POWDER_PLC_INTERLOCK".NCU_TO_POWDER.UNIT_02_POWDER_FEEDER_2_HOPPER_TEMPERATURE_NOMINAL_LINE_1)
   END_RUNG
   RUNG wire#w1
      Move(in := "DB2401_DBB_DEFINE".DBR_244, out1 => "DB7340_POWDER_PLC_INTERLOCK".NCU_TO_POWDER.UNIT_02_POWDER_FEEDER_2_CARRIER_GAS_NOMINAL_LINE_2)
      Move(in := "DB2401_DBB_DEFINE".DBR_252, out1 => "DB7340_POWDER_PLC_INTERLOCK".NCU_TO_POWDER.UNIT_02_POWDER_FEEDER_2_DISK_SPEED_NOMINAL_LINE_2)
      Move(in := "DB2401_DBB_DEFINE".DBR_260, out1 => "DB7340_POWDER_PLC_INTERLOCK".NCU_TO_POWDER.UNIT_02_POWDER_FEEDER_2_STIRRER_SPEED_NOMINAL_LINE_2)
      Move(in := "DB2401_DBB_DEFINE".DBR_268, out1 => "DB7340_POWDER_PLC_INTERLOCK".NCU_TO_POWDER.UNIT_02_POWDER_FEEDER_2_HOPPER_TEMPERATURE_NOMINAL_LINE_2)
   END_RUNG
   // the same network as SCL:
   IF NOT ("M_ONE" AND "DB2001_MODES_GENERAL".GENERAL.MANUAL_SELECTED) THEN
       "DB7340_POWDER_PLC_INTERLOCK".NCU_TO_POWDER.UNIT_02_POWDER_FEEDER_2_CARRIER_GAS_NOMINAL_LINE_1 := "DB2401_DBB_DEFINE".DBR_240;
       "DB7340_POWDER_PLC_INTERLOCK".NCU_TO_POWDER.UNIT_02_POWDER_FEEDER_2_DISK_SPEED_NOMINAL_LINE_1 := "DB2401_DBB_DEFINE".DBR_248;
       "DB7340_POWDER_PLC_INTERLOCK".NCU_TO_POWDER.UNIT_02_POWDER_FEEDER_2_STIRRER_SPEED_NOMINAL_LINE_1 := "DB2401_DBB_DEFINE".DBR_256;
       "DB7340_POWDER_PLC_INTERLOCK".NCU_TO_POWDER.UNIT_02_POWDER_FEEDER_2_HOPPER_TEMPERATURE_NOMINAL_LINE_1 := "DB2401_DBB_DEFINE".DBR_264;
       "DB7340_POWDER_PLC_INTERLOCK".NCU_TO_POWDER.UNIT_02_POWDER_FEEDER_2_CARRIER_GAS_NOMINAL_LINE_2 := "DB2401_DBB_DEFINE".DBR_244;
       "DB7340_POWDER_PLC_INTERLOCK".NCU_TO_POWDER.UNIT_02_POWDER_FEEDER_2_DISK_SPEED_NOMINAL_LINE_2 := "DB2401_DBB_DEFINE".DBR_252;
       "DB7340_POWDER_PLC_INTERLOCK".NCU_TO_POWDER.UNIT_02_POWDER_FEEDER_2_STIRRER_SPEED_NOMINAL_LINE_2 := "DB2401_DBB_DEFINE".DBR_260;
       "DB7340_POWDER_PLC_INTERLOCK".NCU_TO_POWDER.UNIT_02_POWDER_FEEDER_2_HOPPER_TEMPERATURE_NOMINAL_LINE_2 := "DB2401_DBB_DEFINE".DBR_268;
   END_IF;
END_REGION

REGION Network 28: EKS ACCESS LEVELS
   RUNG wire#powerrail
      Contact( "M_ONE" )
      wire#w1
      Move(in := "LTLP_HMIProInterfaceData".currentProtectLevel, out1 => "DB7340_POWDER_PLC_INTERLOCK".NCU_TO_POWDER.CURRENT_PROTECTION_LEVEL)
      Move(in := "LTLP_HMIProInterfaceData".eksOperatorIdentification, out1 => "DB7340_POWDER_PLC_INTERLOCK".NCU_TO_POWDER.EKS_OPERATOR_IDENTIFICATION)
   END_RUNG
   RUNG wire#w1
      Move(in := "LTLP_HMIProInterfaceData".eksIdent1, out1 => "DB7340_POWDER_PLC_INTERLOCK".NCU_TO_POWDER.EKS_IDENT_1)
      Move(in := "LTLP_HMIProInterfaceData".eksIdent2, out1 => "DB7340_POWDER_PLC_INTERLOCK".NCU_TO_POWDER.EKS_IDENT_2)
      Move(in := "LTLP_HMIProInterfaceData".eksIdent3, out1 => "DB7340_POWDER_PLC_INTERLOCK".NCU_TO_POWDER.EKS_IDENT_3)
      Move(in := "LTLP_HMIProInterfaceData".eksIdent4, out1 => "DB7340_POWDER_PLC_INTERLOCK".NCU_TO_POWDER.EKS_IDENT_4)
   END_RUNG
   RUNG wire#w1
      Move(in := "LTLP_HMIProInterfaceData".eksIdent5, out1 => "DB7340_POWDER_PLC_INTERLOCK".NCU_TO_POWDER.EKS_IDENT_5)
      Move(in := "LTLP_HMIProInterfaceData".eksIdent6, out1 => "DB7340_POWDER_PLC_INTERLOCK".NCU_TO_POWDER.EKS_IDENT_6)
      Move(in := "LTLP_HMIProInterfaceData".eksIdent7, out1 => "DB7340_POWDER_PLC_INTERLOCK".NCU_TO_POWDER.EKS_IDENT_7)
      Move(in := "LTLP_HMIProInterfaceData".eksIdent8, out1 => "DB7340_POWDER_PLC_INTERLOCK".NCU_TO_POWDER.EKS_IDENT_8)
   END_RUNG
   // the same network as SCL:
   IF "M_ONE" THEN
       "DB7340_POWDER_PLC_INTERLOCK".NCU_TO_POWDER.CURRENT_PROTECTION_LEVEL := "LTLP_HMIProInterfaceData".currentProtectLevel;
       "DB7340_POWDER_PLC_INTERLOCK".NCU_TO_POWDER.EKS_OPERATOR_IDENTIFICATION := "LTLP_HMIProInterfaceData".eksOperatorIdentification;
       "DB7340_POWDER_PLC_INTERLOCK".NCU_TO_POWDER.EKS_IDENT_1 := "LTLP_HMIProInterfaceData".eksIdent1;
       "DB7340_POWDER_PLC_INTERLOCK".NCU_TO_POWDER.EKS_IDENT_2 := "LTLP_HMIProInterfaceData".eksIdent2;
       "DB7340_POWDER_PLC_INTERLOCK".NCU_TO_POWDER.EKS_IDENT_3 := "LTLP_HMIProInterfaceData".eksIdent3;
       "DB7340_POWDER_PLC_INTERLOCK".NCU_TO_POWDER.EKS_IDENT_4 := "LTLP_HMIProInterfaceData".eksIdent4;
       "DB7340_POWDER_PLC_INTERLOCK".NCU_TO_POWDER.EKS_IDENT_5 := "LTLP_HMIProInterfaceData".eksIdent5;
       "DB7340_POWDER_PLC_INTERLOCK".NCU_TO_POWDER.EKS_IDENT_6 := "LTLP_HMIProInterfaceData".eksIdent6;
       "DB7340_POWDER_PLC_INTERLOCK".NCU_TO_POWDER.EKS_IDENT_7 := "LTLP_HMIProInterfaceData".eksIdent7;
       "DB7340_POWDER_PLC_INTERLOCK".NCU_TO_POWDER.EKS_IDENT_8 := "LTLP_HMIProInterfaceData".eksIdent8;
   END_IF;
END_REGION
END_FUNCTION
